(*			
	RafalOS
	Rafał Osajda		20.11.2025		TC 4024.66
	Moduł przygotowania danych dla Okna receptur we wszsytkich trybach
*)
FUNCTION_BLOCK FB_MCHMIPrepareDataForScreen_02_XX EXTENDS FB_MCHMIPrepareDataForScreen IMPLEMENTS ITF_MCHMIPrepareDataForScreen
VAR
	itfMachineControlHMI	: ITF_MCHMIMachineControl_HMI_PrepScr_02_XX;
	refstData				: REFERENCE TO ST_MCHMIPrepareScreen_02_XX;
END_VAR

(*			
	RafalOS
	Rafał Osajda		19.11.2025		TC 4024.66
	Czyści danych przy zmienia ramki po poprzedniej ramce
*)
METHOD PUBLIC ClearAfterScreen : BOOL
VAR_INPUT
END_VAR
SUPER^.ClearAfterScreen ();
END_METHOD

METHOD PUBLIC LinkDataHMI_02_XX : BOOL
VAR_INPUT
	refstData				: REFERENCE TO ST_MCHMIPrepareScreen_02_XX;
END_VAR
THIS^.refstData REF= refstData;
END_METHOD

METHOD PUBLIC LinkMachineControlHMI : BOOL
VAR_INPUT
	fbMachineControlHMI	: ITF_MCHMIMachineControl_HMI_PrepScr_02_XX;
END_VAR
this^.itfMachineControlHMI := fbMachineControlHMI;
END_METHOD

(*			
	RafalOS
	Rafał Osajda		14.11.2025		TC 4024.66
	Metoda przygotowywania danych dla HMI 
	W niej odbywa się odpytywanie właściego elementu przez łącznik
*)
METHOD PUBLIC PrepareDataForHMI : BOOL
VAR_INPUT
END_VAR




(*	Zewnętrzna obsługa wyświetlania 	*)
SUPER^.PrepareDataForHMI ();
END_METHOD

(*			
	RafalOS
	Rafał Osajda		19.11.2025		TC 4024.66
	Przygotowanie ramki pood tamke do wyświetlenia - tylko przygotowanie a nie przygotowanie danych do wyświetlenia
*)
METHOD PUBLIC PrepareForScreen : BOOL
VAR_INPUT
END_VAR
SUPER^.PrepareForScreen ();
END_METHOD

END_FUNCTION_BLOCK

(* stored: Version 1.1.0.1
   POU FB_MCHMIPrepareDataForScreen_02_XX: Id {3e345615-3045-0b97-1325-577dd10d4eb7}, SpecialFunc None
   Folder ITF_PDFS: Id {467dd6eb-033b-043b-391b-aaf5e7c85d56}
   Method ClearAfterScreen: Id {769c4d88-7d7c-0abd-3ec8-a2785eba0c8a}
   Method LinkDataHMI_02_XX: Id {b9da66c4-53ca-0131-2aca-8ea6a6948732}
   Method LinkMachineControlHMI: Id {f37cb12b-6b85-01b7-0d56-00458746af91}
   Method PrepareDataForHMI: Id {c0a0e110-4c8c-0f99-36c8-629e7e3d43c4}
   Method PrepareForScreen: Id {53b07278-0656-0582-30f0-5f16589c93c8} *)
